// TIA Portal V18 export
// export: Created 2026-06-08T16:04:36.882519Z, ExportSetting WithDefaults, DisplayName Totally Integrated Automation Portal, DisplayVersion V18, DisplayName TIA Portal Openness, DisplayVersion V18, DisplayName TIA Portal Version Control Interface, DisplayVersion V18, DisplayName STEP 7 Professional, DisplayVersion V18, DisplayName STEP 7 Safety, DisplayVersion V18, DisplayName WinCC Professional, DisplayVersion V18
VAR_GLOBAL   // PLC tag table "PTRIG"
   P1 AT %M330.0 : Bool;
   P2 AT %M330.1 : Bool;
   P3 AT %M330.2 : Bool;
   P4 AT %M330.3 : Bool;
   P5 AT %M330.4 : Bool;
   P6 AT %M330.5 : Bool;
   P7 AT %M330.6 : Bool;
   P8 AT %M330.7 : Bool;
   P9 AT %M331.0 : Bool;
   P10 AT %M331.1 : Bool;
   P11 AT %M331.2 : Bool;
END_VAR
